    TriggL T1773,vl,laserOFF,z0,toolEtna\WObj:=wobjEtna;
    TriggL T1774,v50,laserON,z0,toolEtna\WObj:=wobjEtna;
    TriggL T1775,vl,laserOFF,z0,toolEtna\WObj:=wobjEtna;
    TriggL T1776,v50,laserON,z0,toolEtna\WObj:=wobjEtna;
    TriggL T1777,vl,laserOFF,z0,toolEtna\WObj:=wobjEtna;
    TriggL T1778,v50,laserON,z0,toolEtna\WObj:=wobjEtna;
    TriggL T1779,vl,laserOFF,z0,toolEtna\WObj:=wobjEtna;
    TriggL T1780,v50,laserON,z0,toolEtna\WObj:=wobjEtna;
    TriggL T1781,vl,laserOFF,z0,toolEtna\WObj:=wobjEtna;
    TriggL T1782,v50,laserON,z0,toolEtna\WObj:=wobjEtna;
    TriggL T1783,vl,laserOFF,z0,toolEtna\WObj:=wobjEtna;
    TriggL T1784,v50,laserON,z0,toolEtna\WObj:=wobjEtna;
    TriggL T1785,vl,laserOFF,z0,toolEtna\WObj:=wobjEtna;
    TriggL T1786,v50,laserON,z0,toolEtna\WObj:=wobjEtna;
    TriggL T1787,vl,laserOFF,z0,toolEtna\WObj:=wobjEtna;
    TriggL T1788,v50,laserON,z0,toolEtna\WObj:=wobjEtna;
    TriggL T1789,vl,laserOFF,z0,toolEtna\WObj:=wobjEtna;
    TriggL T1790,v50,laserON,z0,toolEtna\WObj:=wobjEtna;
    TriggL T1791,vl,laserOFF,z0,toolEtna\WObj:=wobjEtna;
    TriggL T1792,v50,laserON,z0,toolEtna\WObj:=wobjEtna;
    TriggL T1793,vl,laserOFF,z0,toolEtna\WObj:=wobjEtna;
    TriggL T1794,v50,laserON,z0,toolEtna\WObj:=wobjEtna;
    TriggL T1795,vl,laserOFF,z0,toolEtna\WObj:=wobjEtna;
    TriggL T1796,v50,laserON,z0,toolEtna\WObj:=wobjEtna;
    TriggL T1797,vl,laserOFF,z0,toolEtna\WObj:=wobjEtna;
    TriggL T1798,v50,laserON,z0,toolEtna\WObj:=wobjEtna;
    TriggL T1799,vl,laserOFF,z0,toolEtna\WObj:=wobjEtna;
    TriggL T1800,v50,laserON,z0,toolEtna\WObj:=wobjEtna;
    TriggL T1801,vl,laserOFF,z0,toolEtna\WObj:=wobjEtna;
    TriggL T1802,v50,laserON,z0,toolEtna\WObj:=wobjEtna;
    TriggL T1803,vl,laserOFF,z0,toolEtna\WObj:=wobjEtna;
    TriggL T1804,v50,laserON,z0,toolEtna\WObj:=wobjEtna;
    TriggL T1805,vl,laserOFF,z0,toolEtna\WObj:=wobjEtna;
    TriggL T1806,v50,laserON,z0,toolEtna\WObj:=wobjEtna;
    TriggL T1807,vl,laserOFF,z0,toolEtna\WObj:=wobjEtna;
    TriggL T1808,v50,laserON,z0,toolEtna\WObj:=wobjEtna;
    TriggL T1809,vl,laserOFF,z0,toolEtna\WObj:=wobjEtna;
    TriggL T1810,v50,laserON,z0,toolEtna\WObj:=wobjEtna;
    TriggL T1811,vl,laserOFF,z0,toolEtna\WObj:=wobjEtna;
    TriggL T1812,v50,laserON,z0,toolEtna\WObj:=wobjEtna;
    TriggL T1813,vl,laserOFF,z0,toolEtna\WObj:=wobjEtna;
    TriggL T1814,v50,laserON,z0,toolEtna\WObj:=wobjEtna;
    TriggL T1815,vl,laserOFF,z0,toolEtna\WObj:=wobjEtna;
    TriggL T1816,v50,laserON,z0,toolEtna\WObj:=wobjEtna;
    TriggL T1817,vl,laserOFF,z0,toolEtna\WObj:=wobjEtna;
    TriggL T1818,v50,laserON,z0,toolEtna\WObj:=wobjEtna;
    TriggL T1819,vl,laserOFF,z0,toolEtna\WObj:=wobjEtna;
    TriggL T1820,v50,laserON,z0,toolEtna\WObj:=wobjEtna;
    TriggL T1821,vl,laserOFF,z0,toolEtna\WObj:=wobjEtna;
    TriggL T1822,v50,laserON,z0,toolEtna\WObj:=wobjEtna;
    TriggL T1823,vl,laserOFF,z0,toolEtna\WObj:=wobjEtna;
    TriggL T1824,v50,laserON,z0,toolEtna\WObj:=wobjEtna;
    TriggL T1825,vl,laserOFF,z0,toolEtna\WObj:=wobjEtna;
    TriggL T1826,v50,laserON,z0,toolEtna\WObj:=wobjEtna;
    TriggL T1827,vl,laserOFF,z0,toolEtna\WObj:=wobjEtna;
    TriggL T1828,v50,laserON,z0,toolEtna\WObj:=wobjEtna;
    TriggL T1829,vl,laserOFF,z0,toolEtna\WObj:=wobjEtna;
    TriggL T1830,v50,laserON,z0,toolEtna\WObj:=wobjEtna;
    TriggL T1831,vl,laserOFF,z0,toolEtna\WObj:=wobjEtna;
    TriggL T1832,v50,laserON,z0,toolEtna\WObj:=wobjEtna;
    TriggL T1833,vl,laserOFF,z0,toolEtna\WObj:=wobjEtna;
    TriggL T1834,v50,laserON,z0,toolEtna\WObj:=wobjEtna;
    TriggL T1835,vl,laserOFF,z0,toolEtna\WObj:=wobjEtna;
    TriggL T1836,v50,laserON,z0,toolEtna\WObj:=wobjEtna;
    TriggL T1837,vl,laserOFF,z0,toolEtna\WObj:=wobjEtna;
    TriggL T1838,v50,laserON,z0,toolEtna\WObj:=wobjEtna;
    TriggL T1839,vl,laserOFF,z0,toolEtna\WObj:=wobjEtna;
    TriggL T1840,v50,laserON,z0,toolEtna\WObj:=wobjEtna;
    TriggL T1841,vl,laserOFF,z0,toolEtna\WObj:=wobjEtna;
    TriggL T1842,v50,laserON,z0,toolEtna\WObj:=wobjEtna;
    TriggL T1843,vl,laserOFF,z0,toolEtna\WObj:=wobjEtna;
    TriggL T1844,v50,laserON,z0,toolEtna\WObj:=wobjEtna;
    TriggL T1845,vl,laserOFF,z0,toolEtna\WObj:=wobjEtna;
    TriggL T1846,v50,laserON,z0,toolEtna\WObj:=wobjEtna;
    TriggL T1847,vl,laserOFF,z0,toolEtna\WObj:=wobjEtna;
    TriggL T1848,v50,laserON,z0,toolEtna\WObj:=wobjEtna;
    TriggL T1849,vl,laserOFF,z0,toolEtna\WObj:=wobjEtna;
    TriggL T1850,v50,laserON,z0,toolEtna\WObj:=wobjEtna;
    TriggL T1851,vl,laserOFF,z0,toolEtna\WObj:=wobjEtna;
    TriggL T1852,v50,laserON,z0,toolEtna\WObj:=wobjEtna;
    TriggL T1853,vl,laserOFF,z0,toolEtna\WObj:=wobjEtna;
    TriggL T1854,v50,laserON,z0,toolEtna\WObj:=wobjEtna;
    TriggL T1855,vl,laserOFF,z0,toolEtna\WObj:=wobjEtna;
    TriggL T1856,v50,laserON,z0,toolEtna\WObj:=wobjEtna;
    TriggL T1857,vl,laserOFF,z0,toolEtna\WObj:=wobjEtna;
    TriggL T1858,v50,laserON,z0,toolEtna\WObj:=wobjEtna;
    TriggL T1859,vl,laserOFF,z0,toolEtna\WObj:=wobjEtna;
    TriggL T1860,v50,laserON,z0,toolEtna\WObj:=wobjEtna;
    TriggL T1861,vl,laserOFF,z0,toolEtna\WObj:=wobjEtna;
    TriggL T1862,v50,laserON,z0,toolEtna\WObj:=wobjEtna;
    TriggL T1863,vl,laserOFF,z0,toolEtna\WObj:=wobjEtna;
    TriggL T1864,v50,laserON,z0,toolEtna\WObj:=wobjEtna;
    TriggL T1865,vl,laserOFF,z0,toolEtna\WObj:=wobjEtna;
    TriggL T1866,v50,laserON,z0,toolEtna\WObj:=wobjEtna;
    TriggL T1867,vl,laserOFF,z0,toolEtna\WObj:=wobjEtna;
    TriggL T1868,v50,laserON,z0,toolEtna\WObj:=wobjEtna;
    TriggL T1869,vl,laserOFF,z0,toolEtna\WObj:=wobjEtna;
    TriggL T1870,v50,laserON,z0,toolEtna\WObj:=wobjEtna;
    TriggL T1871,vl,laserOFF,z0,toolEtna\WObj:=wobjEtna;
    TriggL T1872,v50,laserON,z0,toolEtna\WObj:=wobjEtna;
    TriggL T1873,vl,laserOFF,z0,toolEtna\WObj:=wobjEtna;
    TriggL T1874,v50,laserON,z0,toolEtna\WObj:=wobjEtna;
    TriggL T1875,vl,laserOFF,z0,toolEtna\WObj:=wobjEtna;
    TriggL T1876,v50,laserON,z0,toolEtna\WObj:=wobjEtna;
    TriggL T1877,vl,laserOFF,z0,toolEtna\WObj:=wobjEtna;
    TriggL T1878,v50,laserON,z0,toolEtna\WObj:=wobjEtna;
    TriggL T1879,vl,laserOFF,z0,toolEtna\WObj:=wobjEtna;
    TriggL T1880,v50,laserON,z0,toolEtna\WObj:=wobjEtna;
    TriggL T1881,vl,laserOFF,z0,toolEtna\WObj:=wobjEtna;
    TriggL T1882,v50,laserON,z0,toolEtna\WObj:=wobjEtna;
    TriggL T1883,vl,laserOFF,z0,toolEtna\WObj:=wobjEtna;
    TriggL T1884,v50,laserON,z0,toolEtna\WObj:=wobjEtna;
    TriggL T1885,vl,laserOFF,z0,toolEtna\WObj:=wobjEtna;
    TriggL T1886,v50,laserON,z0,toolEtna\WObj:=wobjEtna;
    TriggL T1887,vl,laserOFF,z0,toolEtna\WObj:=wobjEtna;
    TriggL T1888,v50,laserON,z0,toolEtna\WObj:=wobjEtna;
    TriggL T1889,vl,laserOFF,z0,toolEtna\WObj:=wobjEtna;
    TriggL T1890,v50,laserON,z0,toolEtna\WObj:=wobjEtna;
    TriggL T1891,vl,laserOFF,z0,toolEtna\WObj:=wobjEtna;
    TriggL T1892,v50,laserON,z0,toolEtna\WObj:=wobjEtna;
    TriggL T1893,vl,laserOFF,z0,toolEtna\WObj:=wobjEtna;
    TriggL T1894,v50,laserON,z0,toolEtna\WObj:=wobjEtna;
    TriggL T1895,vl,laserOFF,z0,toolEtna\WObj:=wobjEtna;
    TriggL T1896,v50,laserON,z0,toolEtna\WObj:=wobjEtna;
    TriggL T1897,vl,laserOFF,z0,toolEtna\WObj:=wobjEtna;
    TriggL T1898,v50,laserON,z0,toolEtna\WObj:=wobjEtna;
    TriggL T1899,vl,laserOFF,z0,toolEtna\WObj:=wobjEtna;
    TriggL T1900,v50,laserON,z0,toolEtna\WObj:=wobjEtna;
    TriggL T1901,vl,laserOFF,z0,toolEtna\WObj:=wobjEtna;
    TriggL T1902,v50,laserON,z0,toolEtna\WObj:=wobjEtna;
    TriggL T1903,vl,laserOFF,z0,toolEtna\WObj:=wobjEtna;
    TriggL T1904,v50,laserON,z0,toolEtna\WObj:=wobjEtna;
    TriggL T1905,vl,laserOFF,z0,toolEtna\WObj:=wobjEtna;
    TriggL T1906,v50,laserON,z0,toolEtna\WObj:=wobjEtna;
    TriggL T1907,vl,laserOFF,z0,toolEtna\WObj:=wobjEtna;
    TriggL T1908,v50,laserON,z0,toolEtna\WObj:=wobjEtna;
    TriggL T1909,vl,laserOFF,z0,toolEtna\WObj:=wobjEtna;
    TriggL T1910,v50,laserON,z0,toolEtna\WObj:=wobjEtna;
    TriggL T1911,vl,laserOFF,z0,toolEtna\WObj:=wobjEtna;
    TriggL T1912,v50,laserON,z0,toolEtna\WObj:=wobjEtna;
    TriggL T1913,vl,laserOFF,z0,toolEtna\WObj:=wobjEtna;
    TriggL T1914,v50,laserON,z0,toolEtna\WObj:=wobjEtna;
    TriggL T1915,vl,laserOFF,z0,toolEtna\WObj:=wobjEtna;
    TriggL T1916,v50,laserON,z0,toolEtna\WObj:=wobjEtna;
    TriggL T1917,vl,laserOFF,z0,toolEtna\WObj:=wobjEtna;
    TriggL T1918,v50,laserON,z0,toolEtna\WObj:=wobjEtna;
    TriggL T1919,vl,laserOFF,z0,toolEtna\WObj:=wobjEtna;
    TriggL T1920,v50,laserON,z0,toolEtna\WObj:=wobjEtna;
    TriggL T1921,vl,laserOFF,z0,toolEtna\WObj:=wobjEtna;

    Reset doLDLStartST;
ENDPROC

PROC mainEtna()
    Set doLDLExtern;
    Set doLDLRequest;
    Set doLDLLaserON;
    WaitDI diLDLLaserON,1;
    Set doLDLStandBy;

    SetGO GoLDL_Prog, 5;
    WaitTime 1;
    SetGO GoLDL_Pwr3, 1100;

    TriggIO laserON, 0\DOp:=doLDLStartST, 1;
    TriggIO laserOFF, 0\DOp:=doLDLStartST, 0;

    Set DoWeldGas;
    !MedicoatL2 "OFF", 5, 20, 7.5;
    MedicoatL1 "OFF", 5, 20, 15;

    MoveJ [[0.0,0.0,100.0],[0.0,0.0,1.0,0.0],[0,0,-1,0],[9E+09,9E+09,9E+09,9E+09,9E+09,9E+09]],v80,z0,toolEtna\WObj:=wobjEtna;

    ConfL \Off;

    cladding;

    MoveJ [[0.0,0.0,100.0],[0.0,0.0,1.0,0.0],[0,0,-1,0],[9E+09,9E+09,9E+09,9E+09,9E+09,9E+09]],v80,z0,toolEtna\WObj:=wobjEtna;

    Reset doMdtPL2On;
    Reset doMdtPL1On;
    Reset DoWeldGas;

    Reset doLDLStandBy;
    Reset doLDLLaserON;
    Reset doLDLRequest;
    Reset doLDLExtern;

ENDPROC

ENDMODULE
